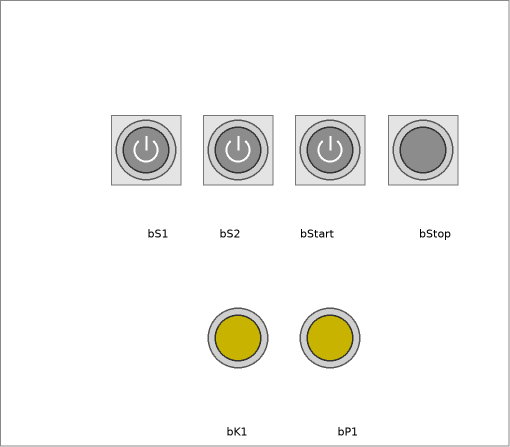
VISUALIZATION Visu  // 510x447
    PowerSwitch (111,115 70x70), variable: MAIN.bS1, behaviour: TOGGLE, style: Switch-PowerSwitch-Gray
    PowerSwitch (203,115 70x70), variable: MAIN.bS2, behaviour: TOGGLE, style: Switch-PowerSwitch-Gray
    PowerSwitch (295,115 70x70), variable: MAIN.bStart, behaviour: TOGGLE, style: Switch-PowerSwitch-Gray
    PushSwitch (388,115 70x70), variable: MAIN.bStop, behaviour: TOGGLE, style: Switch-PushSwitch-Gray
    Lamp1 (203,303 70x70), variable: MAIN.bK1, style: Lamp-Lamp1-Yellow
    Lamp1 (295,303 70x70), variable: MAIN.bP1, style: Lamp-Lamp1-Yellow
    Label (83,219 150x30), "bS1"
    Label (155,219 150x30), "bS2"
    Label (242,219 150x30), "bStart"
    Label (360,219 150x30), "bStop"
    Label (162,417 150x30), "bK1"
    Label (273,417 150x30), "bP1"
END_VISUALIZATION

(* stored: Version 1.1.0.1, ProductVersion 3.1.4024.12
   Visu Visu: Id {62305090-c481-45c6-b846-bc08c238d17e} *)
